(* CoDeSys 2.3.9.28 project: PrahaByt.pro *)
(* Libraries: Y:\Documents\WAGO\Library\Visu_Scheduler_03_e.lib 15.3.11 07:49:24, WagoLibDaylightSaving.lib 2.12.10 14:48:32, DaylightSaving.lib 2.12.10 14:48:32, SysLibRtc.lib 2.12.10 14:48:32, mod_com.lib 2.12.10 14:48:32, SysLibSockets.lib 10.2.11 09:20:54, SysLibFile.lib 2.12.10 14:48:34, SYSLIBTIME.LIB 2.12.10 14:48:32, SysLibMem.lib 2.12.10 14:48:34, Standard.lib 2.12.10 14:48:34, SYSLIBCALLBACK.LIB 2.12.10 14:48:32, Y:\Documents\WAGO\Library\Scheduler_03.lib 9.3.11 15:45:22 *)

(* PLC configuration (modules and I/O channels)
OUT1 AT %QX0.0 [BOOLOnX_Q] Aku. topeni
OUT2 AT %QX0.1 [BOOLOnX_Q] Tiskarna
OUT3 AT %QX0.2 [BOOLOnX_Q] Zasuvka2
OUT4 AT %QX0.3 [BOOLOnX_Q] Zasuvka3
OUT5 AT %QX0.4 [BOOLOnX_Q] Ch_5 Digital output
OUT6 AT %QX0.5 [BOOLOnX_Q] Ch_6 Digital output
OUT7 AT %QX0.6 [BOOLOnX_Q] Ch_7 Digital output
OUT8 AT %QX0.7 [BOOLOnX_Q] Ch_8 Digital output
IN1 AT %IX4.0 [BOOLOnX_I] Nocní proud
IN2 AT %IX4.1 [BOOLOnX_I] Ch_2 Digital input
IN3 AT %IX4.2 [BOOLOnX_I] Ch_3 Digital input
IN4 AT %IX4.3 [BOOLOnX_I] Ch_4 Digital input
IN5 AT %IX4.4 [BOOLOnX_I] Ch_5 Digital input
IN6 AT %IX4.5 [BOOLOnX_I] Ch_6 Digital input
IN7 AT %IX4.6 [BOOLOnX_I] Ch_7 Digital input
IN8 AT %IX4.7 [BOOLOnX_I] Ch_8 Digital input
T1 AT %IW0 [INTOnW_I] Ch_1 signed Input value
T2 AT %IW1 [INTOnW_I] Ch_2 signed Input value
T3 AT %IW2 [INTOnW_I] Ch_3 signed Input value
T4 AT %IW3 [INTOnW_I] Ch_4 signed Input value
Fieldbus variables [FB_VARS] node 1, in %IB0 out %QB0
Flag variables [FLAG_VARS] node 2, in %IB0 out %QB0
*)

(* Global variable list: Global_Variables *)
VAR_GLOBAL
	NocniProud AT %MX1000.1 : BOOL;
	Tiskarna AT %MX1000.2 : BOOL;
	Zasuvka1 AT %MX1000.3 : BOOL;
	TeplotaVenku AT %MW3516 : REAL;
	TeplotaChotba AT %MW3514 : REAL;
	CasDatumAktualni: DT;
END_VAR
VAR_GLOBAL RETAIN PERSISTENT
	typCasProg1: typScheduleWeekly;
	typCasProg2: typScheduleWeekly;
	typCasProg3: typScheduleWeekly;
	typCasProg4: typScheduleWeekly;
	typCasProg5: typScheduleWeekly;
	typCasProg6: typScheduleWeekly;
	typCasProg7: typScheduleWeekly;
	typCasProg8: typScheduleWeekly;
	typCasProg9: typScheduleWeekly;
	typCasProg10: typScheduleWeekly;
	Leto: BOOL;
	DenvTydnu: BYTE;
	sCasDatumAktualni: STRING;
	Kod: INT:= 1567;
	KodZadany: INT;
	Vstup: BOOL:= FALSE;
END_VAR

(* Global variable list: Koupelna_Variables *)
VAR_GLOBAL
	BojlerProvoz AT %MX1000.5 : BOOL;
	Bojler AT %MX1000.4 : BOOL; (* Ohøev vody v bojleru *)
	BojlerMinuty AT %MW3506 : REAL; (* Jak dlouho má bojler ohøívat vodu *)
	BojlerNaNocniProud AT %MX1000.6 : BOOL := TRUE;
END_VAR

(* Global variable list: Topeni_Global *)
VAR_GLOBAL
	TeplotaAktualni2 AT %MW3512 : REAL; (* Namìøená teplota v 1. místnosti. *)
	TeplotaTopeni1 AT %MW3504 : REAL; (* Teplota topení v 1. místnosti. *)
	PozadovanaTeplota1 AT %MW3500 : REAL := 21; (* Pozadovaná teplota v 1. místnosti. *)
	VetrakAutomat AT %MX1001.0 : BOOL := TRUE;
	Vetrak2Automat AT %MX1001.1 : BOOL := TRUE;
	Topeni1: BOOL; (* Topeni v 1. místnosti. *)
	Vetrak1 AT %MX1000.7 : BOOL; (* Vetrak v 1. mistnosti. *)
	Vetrak2 AT %MX1001.2 : BOOL; (* Vetrak v 2. mistnosti. *)
	Vetrak1Minuty AT %MW3518 : REAL; (* Vetrak v 1. jak dlouho má foukat. *)
	Vetrak2Minuty AT %MW3520 : REAL; (* Vetrak v 2. jak dlouho má foukat. *)
	TeplotaAktualni1 AT %MW3502 : REAL := 10; (* Namìøená teplota v 2. místnosti. *)
	TeplotaTopeni2 AT %MW3510 : REAL;
	PozadovanaTeplota2 AT %MW3508 : REAL := 21.5; (* Pozadovaná teplota v 2. místnosti. *)
	Topeni2: BOOL; (* Topeni v 2. místnosti. *)
	PrumernaTeplota: REAL;
END_VAR

(* POU PLC_PRG, CFC *)
PROGRAM PLC_PRG
VAR
	cas_datum: CurTimeEx;
	System_cas: SysTime64;
	System_datum: SystemTimeDate;
	c: iCOMP;
	ano: INT;
	TON: TON;
	d1: D_klop;
	d2: D_klop;
	d3: D_klop;
	d4: D_klop;
END_VAR
VAR (* helpers for the ST form of the networks *)
	_t81 : BOOL;
	_t80 : BOOL;
END_VAR
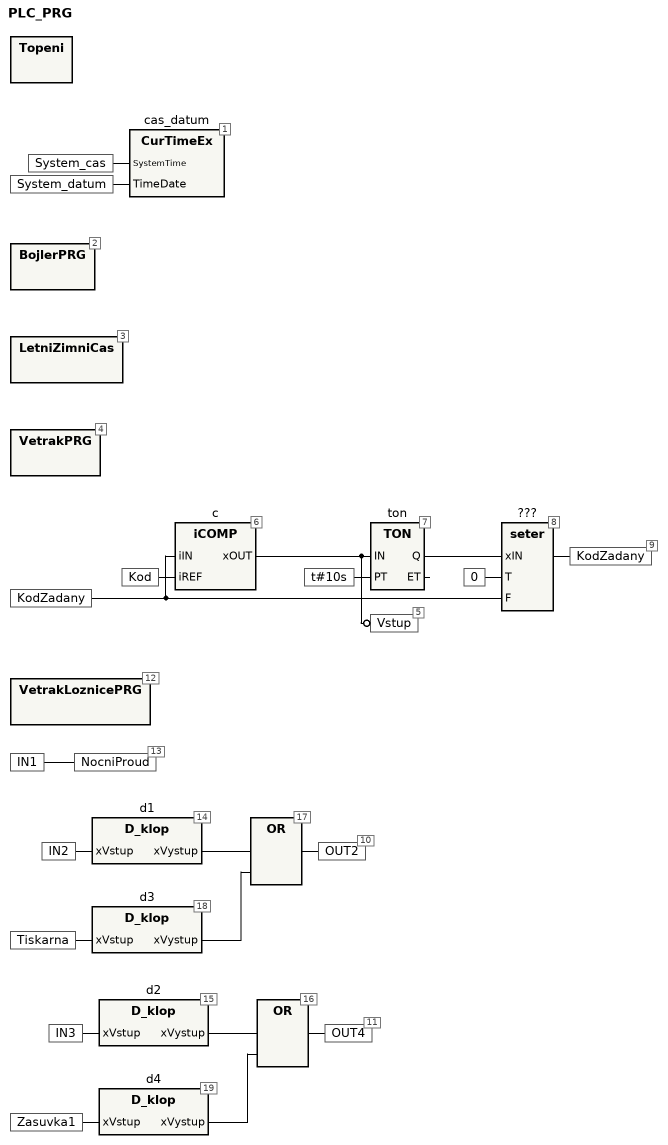
_CFC_ (* Continuous Function Chart, elements in execution order *)
#0 Topeni()
#1 cas_datum:CurTimeEx(SystemTime: System_cas, TimeDate: System_datum)
#2 BojlerPRG()
#3 LetniZimniCas()
#4 VetrakPRG()
#5 Vstup <= NOT #6.xOUT
#6 c:iCOMP(iIN: KodZadany, iREF: Kod)
#7 ton:TON(IN: #6.xOUT, PT: t#10s)
#8 ???:seter(xIN: #7.Q, T: 0, F: KodZadany)
#9 KodZadany <= #8
#10 OUT2 <= #17
#11 OUT4 <= #16
#12 VetrakLoznicePRG()
#13 NocniProud <= IN1
#14 d1:D_klop(xVstup: IN2)
#15 d2:D_klop(xVstup: IN3)
#16 OR(#15.xVystup, #19.xVystup)
#17 OR(#14.xVystup, #18.xVystup)
#18 d3:D_klop(xVstup: Tiskarna)
#19 d4:D_klop(xVstup: Zasuvka1)
_END_CFC_
(* the same logic as Structured Text *)
Topeni();
cas_datum(SystemTime := System_cas, TimeDate := System_datum);
BojlerPRG();
LetniZimniCas();
VetrakPRG();
Vstup := NOT c.xOUT;
c(iIN := KodZadany, iREF := Kod);
ton(IN := c.xOUT, PT := t#10s);
KodZadany := seter(xIN := ton.Q, T := 0, F := KodZadany);
OUT2 := _t81;
OUT4 := _t80;
VetrakLoznicePRG();
NocniProud := IN1;
d1(xVstup := IN2);
d2(xVstup := IN3);
_t80 := d2.xVystup OR d4.xVystup;
_t81 := d1.xVystup OR d3.xVystup;
d3(xVstup := Tiskarna);
d4(xVstup := Zasuvka1);
END_PROGRAM

(* POU Ostatni/iCOMP, ST *)
FUNCTION_BLOCK iCOMP
VAR_INPUT
	iIN: INT;
	iREF: INT;
END_VAR
VAR_OUTPUT
	xOUT: BOOL;

END_VAR
VAR

END_VAR
IF(iIN = iREF)
THEN
	xOUT:= TRUE;
ELSE

	xOUT:= FALSE;
END_IF
END_FUNCTION_BLOCK

(* POU Ostatni/D_klop, ST *)
FUNCTION_BLOCK D_klop
VAR_INPUT
	xVstup: BOOL;
END_VAR
VAR_OUTPUT
	xVystup: BOOL;
END_VAR
VAR
	p: BOOL:= FALSE;
	a: BOOL:= TRUE;
END_VAR
IF(xVstup)
THEN
	IF(p)
	THEN
		IF (a)
			THEN
			xVystup := FALSE;
			p := FALSE;
			a := FALSE;
		END_IF
	ELSE
		IF (a)
			THEN
			xVystup := TRUE;
			p := TRUE;
			a := FALSE;
		END_IF
	END_IF
ELSE
	a:= TRUE;
END_IF
END_FUNCTION_BLOCK

(* POU Topeni, CFC *)
PROGRAM Topeni
VAR
	Spozdeni: TON;
	TO1: TON;
	TO2: TOF;
END_VAR
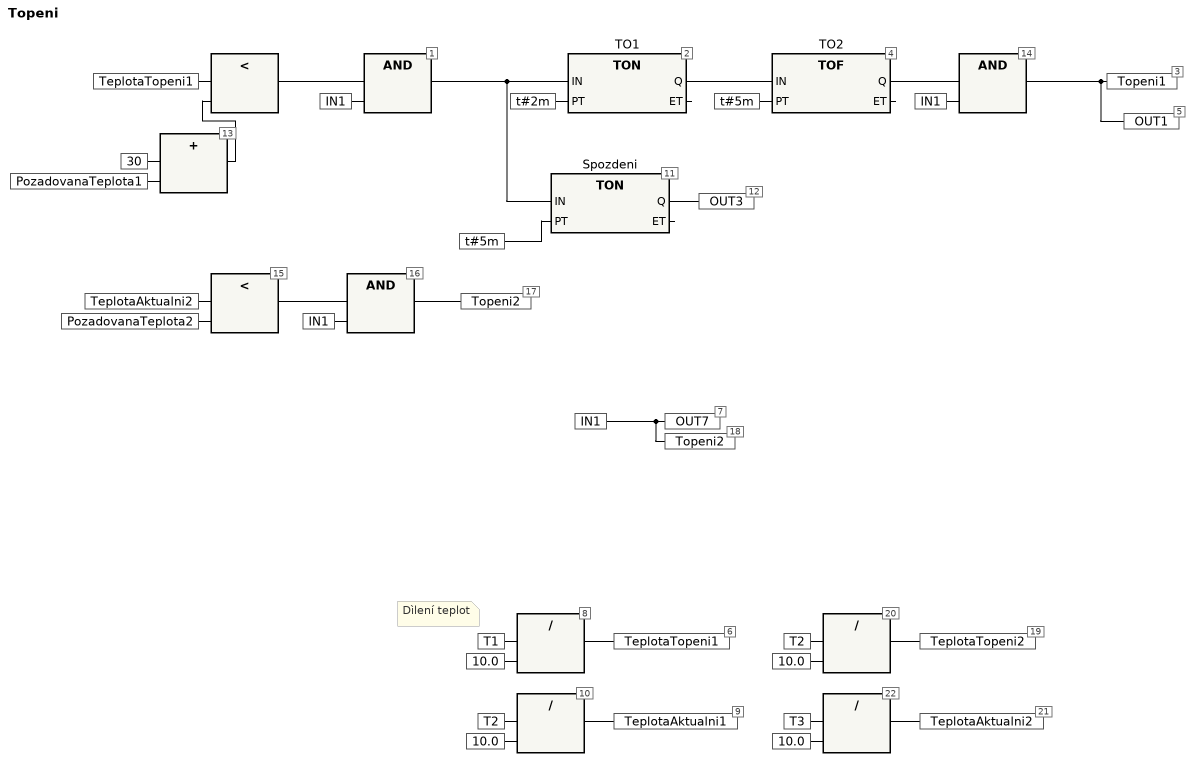
_CFC_ (* Continuous Function Chart, elements in execution order *)
#0 <(TeplotaTopeni1, #13)
#1 AND(#0, IN1)
#2 TO1:TON(IN: #1, PT: t#2m)
#3 Topeni1 <= #14
#4 TO2:TOF(IN: #2.Q, PT: t#5m)
#5 OUT1 <= #14
#6 TeplotaTopeni1 <= #8
(* Dìlení teplot *)
#7 OUT7 <= IN1
#8 /(T1, 10.0)
#9 TeplotaAktualni1 <= #10
#10 /(T2, 10.0)
#11 Spozdeni:TON(IN: #1, PT: t#5m)
#12 OUT3 <= #11.Q
#13 +(30, PozadovanaTeplota1)
#14 AND(#4.Q, IN1)
#15 <(TeplotaAktualni2, PozadovanaTeplota2)
#16 AND(#15, IN1)
#17 Topeni2 <= #16
#18 Topeni2 <= IN1
#19 TeplotaTopeni2 <= #20
#20 /(T2, 10.0)
#21 TeplotaAktualni2 <= #22
#22 /(T3, 10.0)
_END_CFC_
END_PROGRAM

(* POU BojlerPRG, CFC *)
PROGRAM BojlerPRG
VAR
	c1: rCOMP;
	d1: D_klop;
	t: TIME;
	TOF: TOF;
	casovac1: FbScheduleWeekly;
	casovac2: FbScheduleWeekly;
END_VAR
VAR (* helpers for the ST form of the networks *)
	_t2 : BOOL;
	_t17 : BOOL;
	_t3 : BOOL;
	_t11 : TIME;
END_VAR
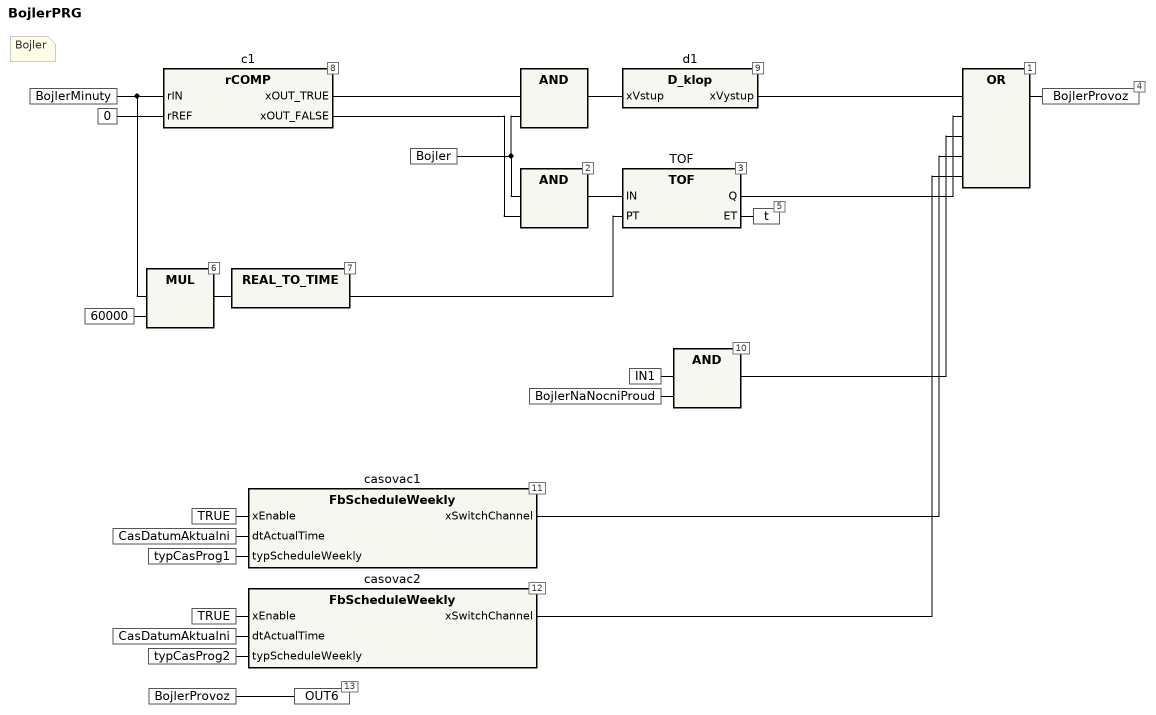
_CFC_ (* Continuous Function Chart, elements in execution order *)
(* Bojler *)
#0 AND(#8.xOUT_TRUE, Bojler)
#1 OR(#9.xVystup, #3.Q, #10, #11.xSwitchChannel, #12.xSwitchChannel)
#2 AND(Bojler, #8.xOUT_FALSE)
#3 TOF:TOF(IN: #2, PT: #7)
#4 BojlerProvoz <= #1
#5 t <= #3.ET
#6 MUL(BojlerMinuty, 60000)
#7 REAL_TO_TIME(#6)
#8 c1:rCOMP(rIN: BojlerMinuty, rREF: 0)
#9 d1:D_klop(xVstup: #0)
#10 AND(IN1, BojlerNaNocniProud)
#11 casovac1:FbScheduleWeekly(xEnable: TRUE, dtActualTime: CasDatumAktualni, typScheduleWeekly: typCasProg1)
#12 casovac2:FbScheduleWeekly(xEnable: TRUE, dtActualTime: CasDatumAktualni, typScheduleWeekly: typCasProg2)
#13 OUT6 <= BojlerProvoz
_END_CFC_
(* the same logic as Structured Text *)
(* Bojler *)
_t2 := c1.xOUT_TRUE AND Bojler;
_t3 := d1.xVystup OR TOF.Q OR _t17 OR casovac1.xSwitchChannel OR casovac2.xSwitchChannel;
TOF(IN := Bojler AND c1.xOUT_FALSE, PT := _t11);
BojlerProvoz := _t3;
t := TOF.ET;
_t11 := REAL_TO_TIME(BojlerMinuty * 60000);
c1(rIN := BojlerMinuty, rREF := 0);
d1(xVstup := _t2);
_t17 := IN1 AND BojlerNaNocniProud;
casovac1(xEnable := TRUE, dtActualTime := CasDatumAktualni, typScheduleWeekly := typCasProg1);
casovac2(xEnable := TRUE, dtActualTime := CasDatumAktualni, typScheduleWeekly := typCasProg2);
OUT6 := BojlerProvoz;
END_PROGRAM

(* POU Ostatni/rCOMP, ST *)
FUNCTION_BLOCK rCOMP
VAR_INPUT
	rIN: REAL;
	rREF: REAL;
END_VAR
VAR_OUTPUT
	xOUT_TRUE: BOOL;
	xOUT_FALSE: BOOL;
END_VAR
VAR

END_VAR
IF(rIN = rREF)
THEN
	xOUT_TRUE:= TRUE;
	xOUT_FALSE:= FALSE;
ELSE
	xOUT_FALSE:= TRUE;
	xOUT_TRUE:= FALSE;
END_IF
END_FUNCTION_BLOCK

(* POU Ostatni/LetniZimniCas, FBD *)
PROGRAM LetniZimniCas
VAR
	sCasDatumPomoc: STRING;
END_VAR
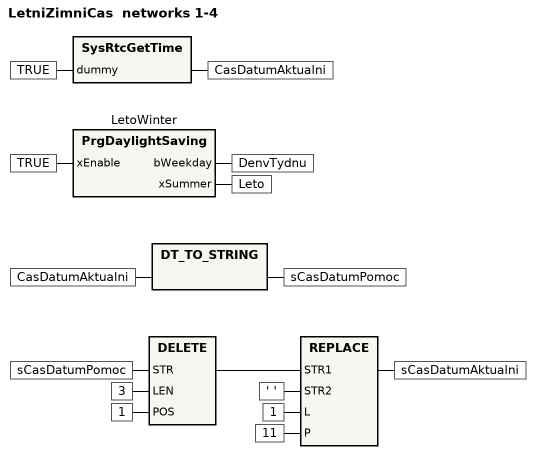
_FBD_ (* Function Block Diagram *)
NETWORK 1 (* Prwcti aktualni datum v procesoru *)
	SysRtcGetTime(dummy: TRUE) => CasDatumAktualni
NETWORK 2 (* Automaticky prechod z letniho na zimni cas / DenvTydnu: Pondeli = 1; Utery = 2; Streda = 3; Ctvrtek = 4; Patek = 5; Sobota = 6; Nedele = 7 *)
	LetoWinter:PrgDaylightSaving(xEnable: TRUE, xSummer => Leto) => DenvTydnu
NETWORK 3
	DT_TO_STRING(CasDatumAktualni) => sCasDatumPomoc
NETWORK 4
	REPLACE(STR1: DELETE(STR: sCasDatumPomoc, LEN: 3, POS: 1), STR2: ' ', L: 1, P: 11) => sCasDatumAktualni
_END_FBD_
(* the same logic as Structured Text *)
(* Network 1: Prwcti aktualni datum v procesoru *)
CasDatumAktualni := SysRtcGetTime(dummy := TRUE);
(* Network 2: Automaticky prechod z letniho na zimni cas / DenvTydnu: Pondeli = 1; Utery = 2; Streda = 3; Ctvrtek = 4; Patek = 5; Sobota = 6; Nedele = 7 *)
LetoWinter(xEnable := TRUE);
Leto := LetoWinter.xSummer;
DenvTydnu := LetoWinter.bWeekday;
(* Network 3 *)
sCasDatumPomoc := DT_TO_STRING(CasDatumAktualni);
(* Network 4 *)
sCasDatumAktualni := REPLACE(DELETE(sCasDatumPomoc, 3, 1), ' ', 1, 11);
END_PROGRAM

(* POU VetrakPRG, CFC *)
PROGRAM VetrakPRG
VAR
	casovac1: FbScheduleWeekly;
	casovac2: FbScheduleWeekly;
	casovac3: FbScheduleWeekly;
	casovac4: FbScheduleWeekly;
	c1: rCOMP;
	d1: D_klop;
	TOF: TOF;
	T1: TON;
	T2: TOF;
END_VAR
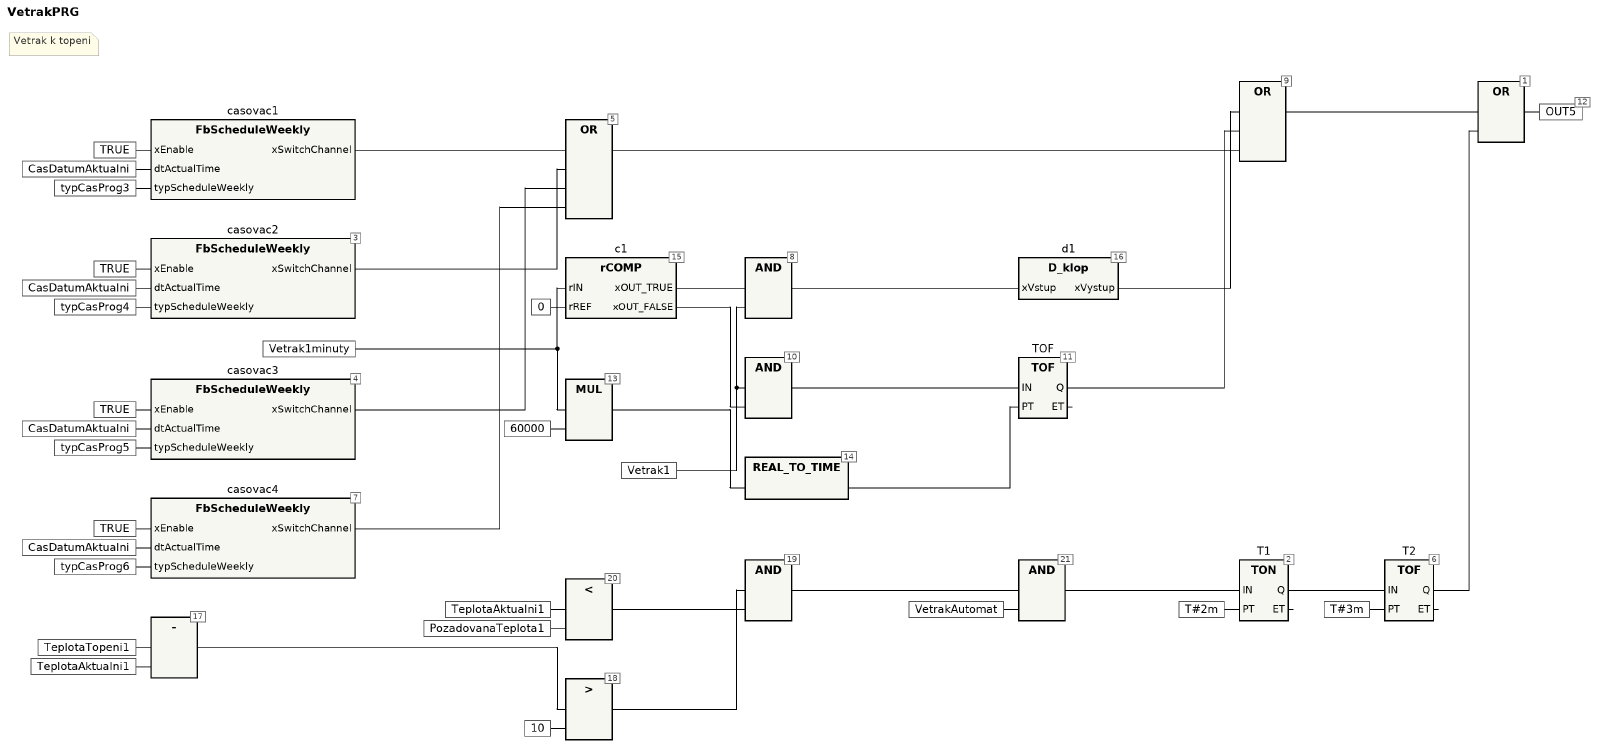
_CFC_ (* Continuous Function Chart, elements in execution order *)
#0 casovac1:FbScheduleWeekly(xEnable: TRUE, dtActualTime: CasDatumAktualni, typScheduleWeekly: typCasProg3)
#1 OR(#9, #6.Q)
#2 T1:TON(IN: #21, PT: T#2m)
#3 casovac2:FbScheduleWeekly(xEnable: TRUE, dtActualTime: CasDatumAktualni, typScheduleWeekly: typCasProg4)
#4 casovac3:FbScheduleWeekly(xEnable: TRUE, dtActualTime: CasDatumAktualni, typScheduleWeekly: typCasProg5)
#5 OR(#0.xSwitchChannel, #3.xSwitchChannel, #4.xSwitchChannel, #7.xSwitchChannel)
#6 T2:TOF(IN: #2.Q, PT: T#3m)
#7 casovac4:FbScheduleWeekly(xEnable: TRUE, dtActualTime: CasDatumAktualni, typScheduleWeekly: typCasProg6)
(* Vetrak k topeni *)
#8 AND(#15.xOUT_TRUE, Vetrak1)
#9 OR(#16.xVystup, #11.Q, #5)
#10 AND(Vetrak1, #15.xOUT_FALSE)
#11 TOF:TOF(IN: #10, PT: #14)
#12 OUT5 <= #1
#13 MUL(Vetrak1minuty, 60000)
#14 REAL_TO_TIME(#13)
#15 c1:rCOMP(rIN: Vetrak1minuty, rREF: 0)
#16 d1:D_klop(xVstup: #8)
#17 -(TeplotaTopeni1, TeplotaAktualni1)
#18 >(#17, 10)
#19 AND(#18, #20)
#20 <(TeplotaAktualni1, PozadovanaTeplota1)
#21 AND(#19, VetrakAutomat)
_END_CFC_
END_PROGRAM

(* POU Ostatni/seter, ST *)
FUNCTION seter : INT
VAR_INPUT
	xIN: BOOL;
	T: INT;
	F: INT;
END_VAR
VAR
END_VAR
IF(xIN)
THEN
seter := T;
ELSE
seter := F;
END_IF
END_FUNCTION

(* POU VetrakLoznicePRG, CFC *)
PROGRAM VetrakLoznicePRG
VAR
	casovac1: FbScheduleWeekly;
	casovac2: FbScheduleWeekly;
	casovac3: FbScheduleWeekly;
	casovac4: FbScheduleWeekly;
	c1: rCOMP;
	d1: D_klop;
	TOF: TOF;
	T1: TON;
	T2: TOF;
END_VAR
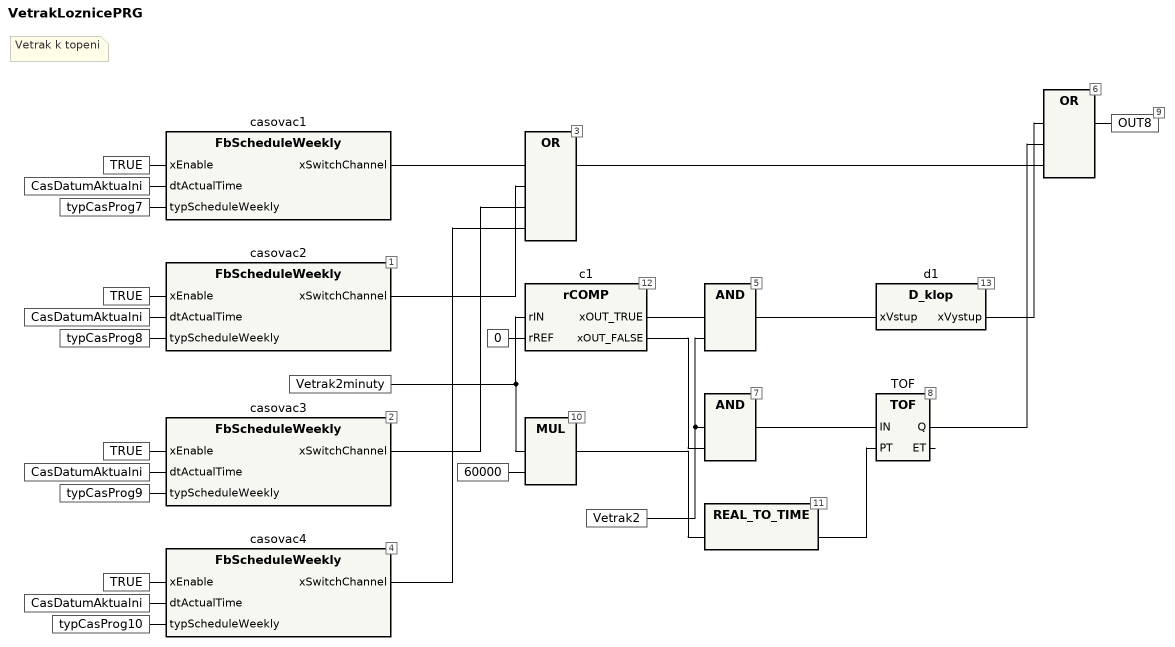
_CFC_ (* Continuous Function Chart, elements in execution order *)
#0 casovac1:FbScheduleWeekly(xEnable: TRUE, dtActualTime: CasDatumAktualni, typScheduleWeekly: typCasProg7)
#1 casovac2:FbScheduleWeekly(xEnable: TRUE, dtActualTime: CasDatumAktualni, typScheduleWeekly: typCasProg8)
#2 casovac3:FbScheduleWeekly(xEnable: TRUE, dtActualTime: CasDatumAktualni, typScheduleWeekly: typCasProg9)
#3 OR(#0.xSwitchChannel, #1.xSwitchChannel, #2.xSwitchChannel, #4.xSwitchChannel)
#4 casovac4:FbScheduleWeekly(xEnable: TRUE, dtActualTime: CasDatumAktualni, typScheduleWeekly: typCasProg10)
(* Vetrak k topeni *)
#5 AND(#12.xOUT_TRUE, Vetrak2)
#6 OR(#13.xVystup, #8.Q, #3)
#7 AND(Vetrak2, #12.xOUT_FALSE)
#8 TOF:TOF(IN: #7, PT: #11)
#9 OUT8 <= #6
#10 MUL(Vetrak2minuty, 60000)
#11 REAL_TO_TIME(#10)
#12 c1:rCOMP(rIN: Vetrak2minuty, rREF: 0)
#13 d1:D_klop(xVstup: #5)
_END_CFC_
END_PROGRAM

(* Visualisation ovladani
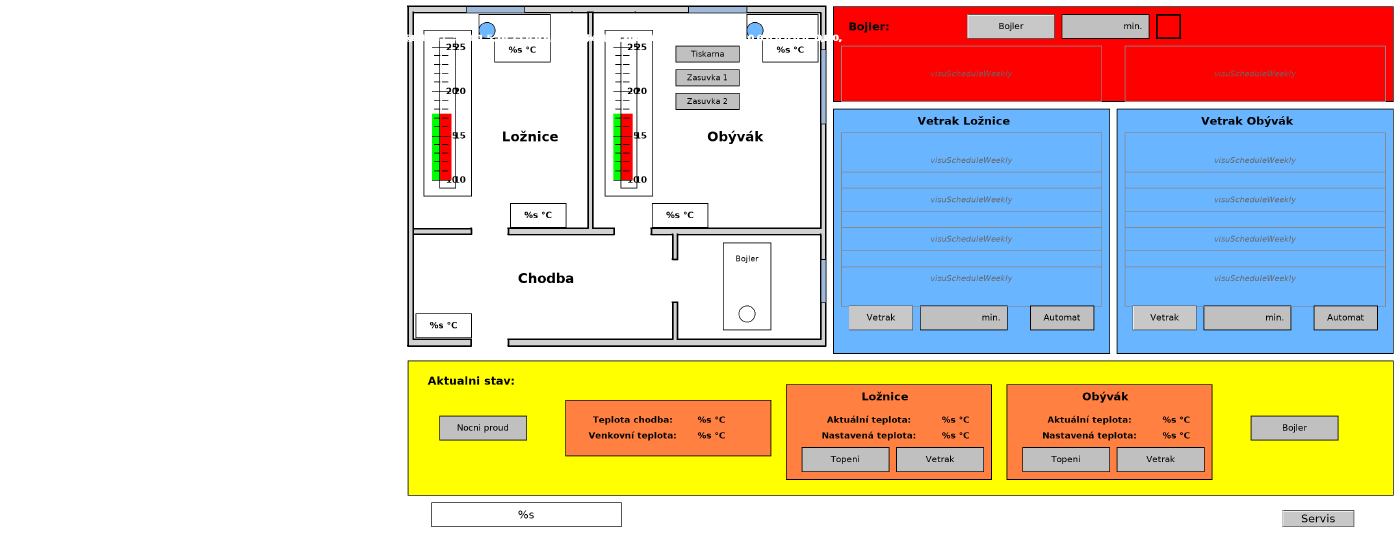
button at (1130,650)-(1221,671): text "Servis"; opens servis
rounded rectangle at (470,50)-(541,81): text "%s °C"; shows .TeplotaTopeni1
rectangle at (50,640)-(291,671): text "%s"; shows .CasDatumAktualni
rounded rectangle at (330,260)-(401,291): text "%s °C"; shows .TeplotaAktualni1
group at (270,50)-(331,241)
  rectangle at (0,0)-(1,1): text "{ExtendedElement},Visu\ElementDLL.ete,1,@Bargraph,61,191,1,1,0,PozadovanaTeplota1,,%.0f,1,5,10,25,0,0,0,0,0,0,0,-13,16,700,Arial,0,255,0,255,0,0,0,0,0,0,0,0,0,,0,0,0,"
  rectangle at (10,95)-(23,178): alarm colour if (PozadovanaTeplota1) < 0; top ((PozadovanaTeplota1 * 1.0) - 17.5)  * -11.0667
  rectangle at (24,167)-(56,188): text "10"
  rectangle at (24,112)-(56,133): text "15"
  rectangle at (24,56)-(56,77): text "20"
  rectangle at (24,1)-(56,22): text "25"
group at (280,50)-(341,241)
  rectangle at (0,0)-(1,1): text "{ExtendedElement},Visu\ElementDLL.ete,1,@Bargraph,61,191,1,1,0,TeplotaAktualni1,,%.0f,1,5,10,25,0,0,0,0,0,0,0,-13,16,700,Arial,255,0,0,255,0,0,0,0,0,0,0,0,0,,0,0,0,"
  rectangle at (10,95)-(23,178): alarm colour if (TeplotaAktualni1) < 0; top ((TeplotaAktualni1 * 1.0) - 17.5)  * -11.0667
  rectangle at (24,167)-(56,188): text "10"
  rectangle at (24,112)-(56,133): text "15"
  rectangle at (24,56)-(56,77): text "20"
  rectangle at (24,1)-(56,22): text "25"
rectangle at (30,470)-(171,501): text "Aktualni stav:"
rounded rectangle at (60,530)-(171,561): text "Nocni proud"; alarm colour if IN1
rounded rectangle at (360,60)-(441,81): text "Tiskarna"; alarm colour if .Tiskarna; toggles .Tiskarna
rounded rectangle at (360,120)-(441,141): text "Zasuvka 2"; alarm colour if .OUT3; toggles .OUT3
rounded rectangle at (360,90)-(441,111): text "Zasuvka 1"; alarm colour if .Zasuvka1; toggles .Zasuvka1
rectangle at (630,140)-(821,171): text "Vetrak Ložnice"
rounded rectangle at (670,390)-(781,421): tooltip 0 = stiskem zapni/ stiskem vypni
rounded rectangle at (740,390)-(781,421): text "min."; tooltip 0 = stiskem zapni/ stiskem vypni
embedded screen at (570,170)-(901,241): visuScheduleWeekly
embedded screen at (570,270)-(901,341): visuScheduleWeekly
embedded screen at (570,220)-(901,291): visuScheduleWeekly
embedded screen at (570,320)-(901,391): visuScheduleWeekly
rectangle at (570,20)-(641,51): text "Bojler:"
rounded rectangle at (850,20)-(961,51): tooltip 0 = stiskem zapni/ stiskem vypni
rounded rectangle at (920,20)-(961,51): text "min."; tooltip 0 = stiskem zapni/ stiskem vypni
rounded rectangle at (970,20)-(1001,51): alarm colour if BojlerNaNocniProud; toggles BojlerNaNocniProud; tooltip èervená = vypnuto; zelená = topí s noèním proudem
embedded screen at (570,60)-(901,131): visuScheduleWeekly
embedded screen at (930,60)-(1261,131): visuScheduleWeekly
rounded rectangle at (1090,530)-(1201,561): text "Bojler"; alarm colour if OUT6
rounded rectangle at (640,570)-(751,601): text "Vetrak"; alarm colour if OUT5
button at (730,20)-(841,51): text "Bojler"; taps Bojler
button at (580,390)-(661,421): text "Vetrak"; taps Vetrak2
ellipse at (440,390)-(461,411): alarm colour if OUT6; taps Bojler
rectangle at (420,320)-(481,341): text "Bojler"
rounded rectangle at (520,570)-(631,601): text "Topeni"; alarm colour if OUT1
rounded rectangle at (450,20)-(541,51): alarm colour if OUT1
ellipse at (450,30)-(471,51): alarm colour if OUT5
rounded rectangle at (810,390)-(891,421): text "Automat"; alarm colour if .Vetrak2Automat; toggles .Vetrak2Automat
rectangle at (520,520)-(691,551): text "Aktuální teplota:"
rectangle at (680,520)-(751,551): text "%s °C"; shows .TeplotaAktualni2
rectangle at (520,540)-(691,571): text "Nastavená teplota:"
rectangle at (680,540)-(751,571): text "%s °C"; shows .PozadovanaTeplota2
rectangle at (560,490)-(691,521): text "Ložnice"
rounded rectangle at (920,570)-(1031,601): text "Vetrak"; alarm colour if OUT5
rounded rectangle at (800,570)-(911,601): text "Topeni"; alarm colour if OUT1
rectangle at (800,520)-(971,551): text "Aktuální teplota:"
rectangle at (960,520)-(1031,551): text "%s °C"; shows .TeplotaAktualni1
rectangle at (800,540)-(971,571): text "Nastavená teplota:"
rectangle at (960,540)-(1031,571): text "%s °C"; shows .PozadovanaTeplota1
rectangle at (840,490)-(971,521): text "Obývák"
rectangle at (220,520)-(391,551): text "Teplota chodba:"
rectangle at (370,520)-(441,551): text "%s °C"; shows .TeplotaChotba
rectangle at (220,540)-(391,571): text "Venkovní teplota:"
rectangle at (370,540)-(441,571): text "%s °C"; shows .TeplotaVenku
rectangle at (110,160)-(241,191): text "Ložnice"
rectangle at (370,160)-(501,191): text "Obývák"
rectangle at (990,140)-(1181,171): text "Vetrak Obývák"
rounded rectangle at (1030,390)-(1141,421): tooltip 0 = stiskem zapni/ stiskem vypni
rounded rectangle at (1100,390)-(1141,421): text "min."; tooltip 0 = stiskem zapni/ stiskem vypni
embedded screen at (930,170)-(1261,241): visuScheduleWeekly
embedded screen at (930,270)-(1261,341): visuScheduleWeekly
embedded screen at (930,220)-(1261,291): visuScheduleWeekly
embedded screen at (930,320)-(1261,391): visuScheduleWeekly
button at (940,390)-(1021,421): text "Vetrak"; taps Vetrak1
rounded rectangle at (1170,390)-(1251,421): text "Automat"; alarm colour if .VetrakAutomat; toggles .VetrakAutomat
rounded rectangle at (110,20)-(201,51): alarm colour if OUT1
ellipse at (110,30)-(131,51): alarm colour if OUT8
rounded rectangle at (130,50)-(201,81): text "%s °C"; shows .TeplotaTopeni2
rounded rectangle at (150,260)-(221,291): text "%s °C"; shows .TeplotaAktualni2
group at (40,50)-(101,241)
  rectangle at (0,0)-(1,1): text "{ExtendedElement},Visu\ElementDLL.ete,1,@Bargraph,61,191,1,1,0,PozadovanaTeplota2,,%.0f,1,5,10,25,0,0,0,0,0,0,0,-13,16,700,Arial,0,255,0,255,0,0,0,0,0,0,0,0,0,,0,0,0,"
  rectangle at (10,95)-(23,178): alarm colour if (PozadovanaTeplota2) < 0; top ((PozadovanaTeplota2 * 1.0) - 17.5)  * -11.0667
  rectangle at (24,167)-(56,188): text "10"
  rectangle at (24,112)-(56,133): text "15"
  rectangle at (24,56)-(56,77): text "20"
  rectangle at (24,1)-(56,22): text "25"
group at (50,50)-(111,241)
  rectangle at (0,0)-(1,1): text "{ExtendedElement},Visu\ElementDLL.ete,1,@Bargraph,61,191,1,1,0,TeplotaAktualni2,,%.0f,1,5,10,25,0,0,0,0,0,0,0,-13,16,700,Arial,255,0,0,255,0,0,0,0,0,0,0,0,0,,0,0,0,"
  rectangle at (10,95)-(23,178): alarm colour if (TeplotaAktualni2) < 0; top ((TeplotaAktualni2 * 1.0) - 17.5)  * -11.0667
  rectangle at (24,167)-(56,188): text "10"
  rectangle at (24,112)-(56,133): text "15"
  rectangle at (24,56)-(56,77): text "20"
  rectangle at (24,1)-(56,22): text "25"
rounded rectangle at (30,400)-(101,431): text "%s °C"; shows .TeplotaChotba
rectangle at (130,340)-(261,371): text "Chodba"
83 more shapes without text or variables
5 elements of other kinds (tables, trends, ...) not read
*)

(* Visualisation plc_visu
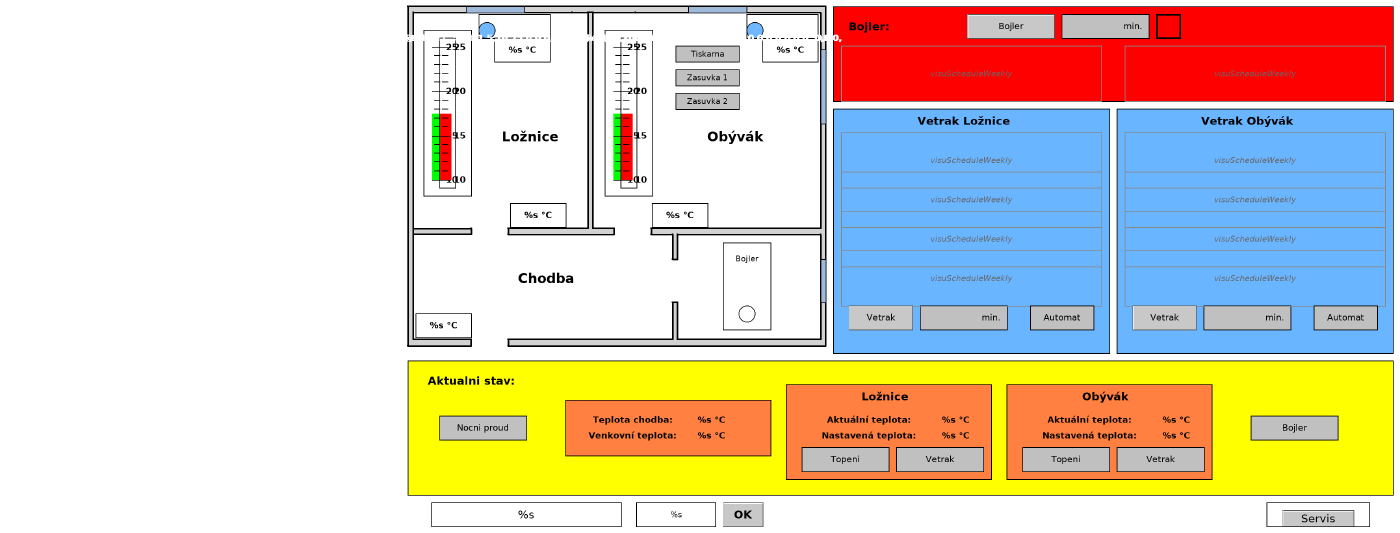
embedded screen at (0,0)-(1271,671): ovladani
rectangle at (310,640)-(411,671): text "%s"; shows KodZadany; editable
button at (420,640)-(471,671): text "OK"; invisible if Vstup; opens ovladani
2 more shapes without text or variables
*)

(* Visualisation servis
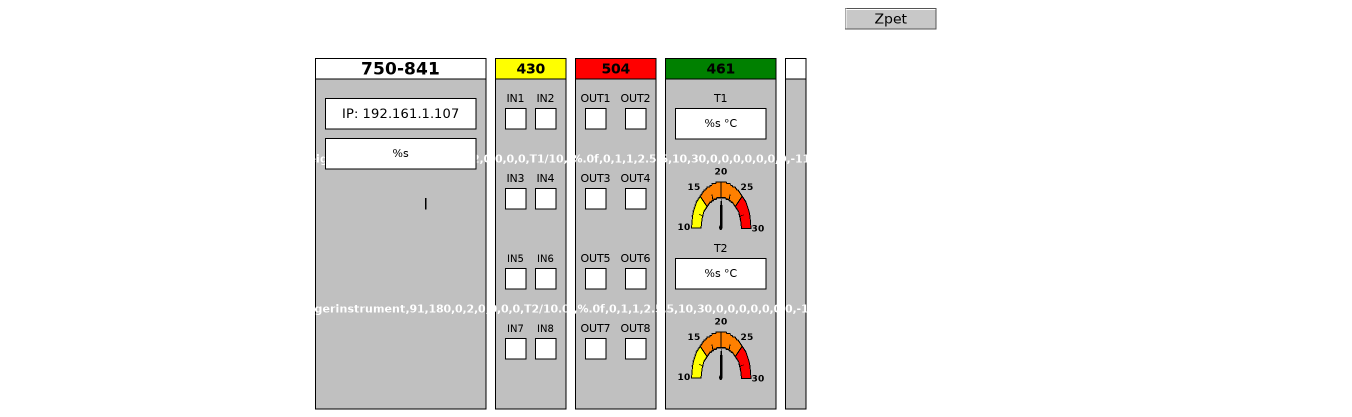
rectangle at (270,60)-(351,81): text "504"
rectangle at (190,60)-(261,81): text "430"
rectangle at (360,60)-(471,81): text "461"
rectangle at (10,60)-(181,81): text "750-841"
rectangle at (20,100)-(171,131): text "IP: 192.161.1.107"
rectangle at (280,110)-(301,131): alarm colour if OUT1; toggles OUT1
rectangle at (270,90)-(311,111): text "OUT1"
rectangle at (320,110)-(341,131): alarm colour if OUT2; toggles OUT2
rectangle at (310,90)-(351,111): text "OUT2"
rectangle at (280,270)-(301,291): alarm colour if OUT5; toggles OUT5
rectangle at (270,250)-(311,271): text "OUT5"
rectangle at (320,270)-(341,291): alarm colour if OUT6; toggles OUT6
rectangle at (310,250)-(351,271): text "OUT6"
rectangle at (200,110)-(221,131): alarm colour if IN1
rectangle at (190,90)-(231,111): text "IN1"
rectangle at (230,110)-(251,131): alarm colour if IN2
rectangle at (220,90)-(261,111): text "IN2"
rectangle at (200,270)-(221,291): alarm colour if IN5
rectangle at (190,250)-(231,271): text "IN5"
rectangle at (230,270)-(251,291): alarm colour if IN6
rectangle at (220,250)-(261,271): text "IN6"
rectangle at (200,190)-(221,211): alarm colour if IN3
rectangle at (190,170)-(231,191): text "IN3"
rectangle at (230,190)-(251,211): alarm colour if IN4
rectangle at (220,170)-(261,191): text "IN4"
rectangle at (200,340)-(221,361): alarm colour if IN8
rectangle at (190,320)-(231,341): text "IN7"
rectangle at (230,340)-(251,361): alarm colour if IN8
rectangle at (220,320)-(261,341): text "IN8"
rectangle at (370,110)-(461,141): text "%s °C"; shows T1/10.0
rectangle at (370,260)-(461,291): text "%s °C"; shows T2/10.0
rectangle at (360,90)-(471,111): text "T1"
rectangle at (360,240)-(471,261): text "T2"
group at (370,160)-(461,241)
  rectangle at (0,0)-(1,1): text "{ExtendedElement},Visu\ElementDLL.ete,0,@Zeigerinstrument,91,180,0,2,0,0,0,0,T1/10,,%.0f,0,1,1,2.5,5,10,30,0,0,0,0,0,0,0,-11,80,700,Arial,1,3,10,15,255,255,0,15,25,255,128,0,25,30,255,0,0,0,255,255,255,,0,0,0,"
  rectangle at (1,38)-(17,52): text "10"
  rectangle at (11,12)-(27,26): text "15"
  rectangle at (38,2)-(54,16): text "20"
  rectangle at (64,12)-(80,26): text "25"
  rectangle at (75,39)-(91,53): text "30"
  polygon at (45,27)-(47,46): angle ((T1/10 * 1.0)-20) * 9
group at (370,310)-(461,391)
  rectangle at (0,0)-(1,1): text "{ExtendedElement},Visu\ElementDLL.ete,0,@Zeigerinstrument,91,180,0,2,0,0,0,0,T2/10.0,,%.0f,0,1,1,2.5,5,10,30,0,0,0,0,0,0,0,-11,80,700,Arial,1,3,10,15,255,255,0,15,25,255,128,0,25,30,255,0,0,0,255,255,255,,0,0,0,"
  rectangle at (1,38)-(17,52): text "10"
  rectangle at (11,12)-(27,26): text "15"
  rectangle at (38,2)-(54,16): text "20"
  rectangle at (64,12)-(80,26): text "25"
  rectangle at (75,39)-(91,53): text "30"
  polygon at (45,27)-(47,46): angle ((T2/10.0 * 1.0)-20) * 9
rectangle at (280,190)-(301,211): alarm colour if OUT3; toggles OUT3
rectangle at (270,170)-(311,191): text "OUT3"
rectangle at (320,190)-(341,211): alarm colour if OUT4; toggles OUT4
rectangle at (310,170)-(351,191): text "OUT4"
rectangle at (280,340)-(301,361): alarm colour if OUT7; toggles OUT7
rectangle at (270,320)-(311,341): text "OUT7"
rectangle at (320,340)-(341,361): alarm colour if OUT8; toggles OUT8
rectangle at (310,320)-(351,341): text "OUT8"
button at (540,10)-(631,31): text "Zpet"; opens plc_visu
rectangle at (20,140)-(171,171): text "%s"; shows .CasDatumAktualni
37 more shapes without text or variables
*)
